{attribute 'qualified_only'}
{attribute 'strict'}
TYPE En_DistanceMode :
(
	Default := 0,
	NearerIsHigher,
	NearerIsLower
);
END_TYPE

(* stored: Version 1.1.0.1, ProductVersion 3.1.4024.9
   DUT En_DistanceMode: Id {36986fab-1f1a-428f-9e67-6bc6eb0e702b} *)
